INTERFACE I_RpcHeaderAccessor

PROPERTY PUBLIC ContentType_Json : T_MAXSTRING
GET
END_GET
END_PROPERTY

METHOD PUBLIC TryGetAcceptResponseFormatFromRequest : BOOL
VAR_INPUT
	Request : I_Request;
	Destination : ANY;
END_VAR
END_METHOD

METHOD PUBLIC TryGetContentTypeFromRequest : BOOL
VAR_INPUT
	Request : I_Request;
	Destination : ANY;
END_VAR
END_METHOD

METHOD PUBLIC TryGetMethodNameFromRequest : BOOL
VAR_INPUT
	Request : I_Request;
	Destination : ANY;
END_VAR
END_METHOD

METHOD PUBLIC TryGetTypeFromRequest : BOOL
VAR_INPUT
	Request : I_Request;
	Destination : ANY;
END_VAR
END_METHOD

END_INTERFACE

(* stored: Version 1.1.0.1, ProductVersion 3.1.4024.12
   Itf I_RpcHeaderAccessor: Id {6414b0e5-9074-0b26-03d1-a04f0b89079c}
   Property ContentType_Json: Id {ffaae006-0a92-01ea-18b6-79163d0161fc}
   Get Get: Id {51bcc622-d17a-06b1-3ead-130353ea8005}
   Method TryGetAcceptResponseFormatFromRequest: Id {d3ae43a2-119f-0a41-107d-2e2ad23b1703}
   Method TryGetContentTypeFromRequest: Id {2f69c95c-26fc-0a8c-1da9-f3f352d247b3}
   Method TryGetMethodNameFromRequest: Id {ac2b8339-0d89-0afc-3b1c-59acdf85cb26}
   Method TryGetTypeFromRequest: Id {ba171ff9-3d29-0ad0-3be8-b1e2e45b0255} *)
